{attribute addProperty BoxType "AT2050-0500-0022"}
{attribute addProperty Id "A_0091_AT2020_5250_0017_AT2020_5250AT2020_C5E5984862678.25"}
{attribute addProperty CRC "1241416301"}
{attribute addProperty SizeInBites "626"}
{attribute addProperty SizeInBytes "78.25"}
TYPE A_0053_AT2050_0500_0022_49FE826D EXTENDS AT2050_BA5A9548 :
STRUCT
	{attribute addProperty Name "A_0091_AT2020_5250_0017_AT2020_5250"}
	A_0091_AT2020_5250_0017_AT2020_5250 : AT2020_C5E59848;
END_STRUCT
END_TYPE

(* stored: Version 1.2.0.0, ProductVersion 3.1.4024.9
   DUT A_0053_AT2050_0500_0022_49FE826D: Id {5ccb9964-7a2c-4ee3-8e82-56fd2bd8525f} *)
